FUNCTION_BLOCK Conveyor1HmiIReq (* Conveyor 1 HMI Interface Requier *)
  (* Standard: 61499-2 *)
  (* Version 0.2, 2003-12-05, JHC, Rockwell Automation, Renamed from NEWCOMPFB. *)
  (* Version 0.1, 2002-01-08, JHC, Rockwell Automation, Added DLY FB as example. *)
  (* Version 0.0, 2000-05-27, JHC, Rockwell Automation *)
  (* Compiler header: package fb.rt.dasdA1.A2.Conveyor; *)
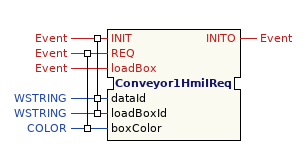
  EVENT_INPUT
    INIT WITH dataId, loadBoxId; (* Initialization Request *)
    REQ WITH boxColor;
    loadBox;
  END_EVENT
  EVENT_OUTPUT
    INITO; (* Initialization Confirm *)
  END_EVENT
  VAR_INPUT
    dataId : WSTRING;
    loadBoxId : WSTRING;
    boxColor : COLOR;
  END_VAR
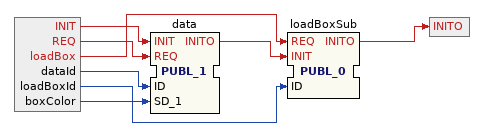
  FBS
    loadBoxSub : PUBL_0;
    data : PUBL_1;
  END_FBS
  EVENT_CONNECTIONS
    loadBox TO loadBoxSub.REQ;
    INIT TO data.INIT;
    REQ TO data.REQ;
    data.INITO TO loadBoxSub.INIT;
    loadBoxSub.INITO TO INITO;
  END_CONNECTIONS
  DATA_CONNECTIONS
    loadBoxId TO loadBoxSub.ID;
    dataId TO data.ID;
    boxColor TO data.SD_1;
  END_CONNECTIONS
END_FUNCTION_BLOCK
